INTERFACE InterfaceVisu

METHOD ZustandsautomatAddVisu : BOOL
VAR_INPUT
	P_Panel						: POINTER TO ST_Panel;
	Name						: STRING(255);
END_VAR
END_METHOD

END_INTERFACE

(* stored: Version 1.1.0.1, ProductVersion 3.1.4024.9
   Itf InterfaceVisu: Id {c3c1a429-7f31-4448-a16e-2db9f68dfc27}
   Method ZustandsautomatAddVisu: Id {0a9bc147-a9d0-48c0-896c-fc9990842c1f} *)
